// TIA Portal V20 export
// export: Created 2025-12-01T14:57:09.6520783Z, ExportSetting None, DisplayName Totally Integrated Automation Portal, DisplayVersion V20 Update 3, DisplayName TIA Portal Openness, DisplayVersion V20 Update 3, DisplayName TIA Portal Version Control Interface, DisplayVersion V20 Update 3, DisplayName STEP 7 Professional, DisplayVersion V20 Update 3, DisplayName STEP 7 Safety, DisplayVersion V20 Update 2, DisplayName WinCC Basic/Comfort/Advanced, DisplayVersion V20 Update 3, DisplayName WinCC Professional, DisplayVersion V20 Update 3, DisplayName WinCC Unified, DisplayVersion V20 Update 3
FUNCTION "FC722_EliminarUT_DeMesa" : Void   // FC722, LAD
TITLE = EliminarUT_DeMesa - Eliminar la UT de la BD
{ S7_Optimized_Access := 'FALSE' }
AUTHOR : TRACKING
NAME : 20130301
VERSION : 3.0
// stored: AutoNumber false, SetENOAutomatically false
   VAR_INPUT
      NumeroUT : UInt;
   END_VAR
   VAR_TEMP
      Mesa : UInt;   // Mesa
      AnteriorUT : UInt;   // UT Anterior
      SiguienteUT : UInt;   // UT Siguiente
      MckeyTemporal : UDInt;   // Para la ordenacion con Mckey
      ColaMckey : UInt;
      ValorReturn : Int;
      Cero : Byte;
   END_VAR
BEGIN

NETWORK
TITLE = Inicilizar
////////////////////////////////////////////////////////////////////////////////
////////////////////////////////////////////////////////////////////////////////
// Inicializa las variables
      L     0;
      T     #AnteriorUT;
      T     #SiguienteUT;



NETWORK
TITLE = Modificar BD de la Mesa -- Previo
////////////////////////////////////////////////////////////////////////////////
////////////////////////////////////////////////////////////////////////////////
////////////////////////////////////////////////////////////////////////////////
// Datos de la UT Mesa, Anterior UT y Siguiente UT
      L     "DB812_UTs_Control".UT[#NumeroUT].MesaActual;
      L     "CTE_OffsetMesa";
      -I;
      T     #Mesa;

      L     "DB812_UTs_Control".UT[#NumeroUT].UT_AnteriorMesa;
      T     #AnteriorUT;
      L     "DB812_UTs_Control".UT[#NumeroUT].UT_SiguienteMesa;
      T     #SiguienteUT;

      L     "DB812_UTs_Control".UT[#NumeroUT].Mckey;
      T     #MckeyTemporal;



////////////////////////////////////////////////////////////////////////////////
// Limpieza de la UT

      L     0;  // Valor a rellenar
      T     #Cero;

// Borrado del DB de los Datos de la UT
      CALL  FILL
      ( BVAL    := #Cero,
        RET_VAL := #ValorReturn,
        BLK     := "DB812_UTs_Control".UT[#NumeroUT]
      );

// Borrado del DB de la Rutas de la UT
      CALL  FILL
      ( BVAL    := #Cero,
        RET_VAL := #ValorReturn,
        BLK     := "DB813_UTs_Ruta".UT[#NumeroUT]
      );

// Borrado del DB de los Datos Auxiliares de la UT
      CALL  FILL
      ( BVAL    := #Cero,
        RET_VAL := #ValorReturn,
        BLK     := "DB814_UTs_Etiqueta".UT[#NumeroUT]
      );
      CALL  FILL
      ( BVAL    := #Cero,
        RET_VAL := #ValorReturn,
        BLK     := "DB815_UTs_Datos".UT[#NumeroUT]
      );
      CALL  FILL
      ( BVAL    := #Cero,
        RET_VAL := #ValorReturn,
        BLK     := "DB816_UTs_TextoPantalla".UT[#NumeroUT]
      );
      CALL  FILL
      ( BVAL    := #Cero,
        RET_VAL := #ValorReturn,
        BLK     := "DB820_UTs_DatosQUBIQA".UT[#NumeroUT]
      );
      CALL  FILL
      ( BVAL    := #Cero,
        RET_VAL := #ValorReturn,
        BLK     := "DB821_UTs_DatosIKPAL".UT[#NumeroUT]
      );



NETWORK
TITLE = -- UT Anterior
////////////////////////////////////////////////////////////////////////////////
////////////////////////////////////////////////////////////////////////////////
////////////////////////////////////////////////////////////////////////////////
// Modificar la UT Anterior
      SET;
      L     #AnteriorUT;
      L     0;
      ==I;  // Era la UT primera de la Mesa
      JC    PrimeraUT_EnColaMesa;
      JU    NoPrimeraUT_EnColaMesa;


////////////////////////////////////////////////////////////////////////////////
// No es la primar UT de la Mesa
NoPrimeraUT_EnColaMesa:NOP   0;
      L     #SiguienteUT;
      T     "DB812_UTs_Control".UT[#AnteriorUT].UT_SiguienteMesa;

      JU    SiguienteUT_EnColaMesa;


////////////////////////////////////////////////////////////////////////////////
// Es la primera UT de la Mesa
PrimeraUT_EnColaMesa:NOP   0;
      L     #SiguienteUT;
      T     "DB810_ColasMesas".Colas[#Mesa].UT_PrimeraMesa;

      JU    SiguienteUT_EnColaMesa;



NETWORK
TITLE = -- UT Siguiente
////////////////////////////////////////////////////////////////////////////////
////////////////////////////////////////////////////////////////////////////////
////////////////////////////////////////////////////////////////////////////////
// Modificar la UT Siguiente
SiguienteUT_EnColaMesa:NOP   0;
      L     #SiguienteUT;
      L     0;
      ==I;
      JC    Final_EnColaDeMesa;  // Era la UT ultima de la Mesa

////////////////////////////////////////////////////////////////////////////////
// No es la Ultima UT de la Mesa
      L     #AnteriorUT;
      T     "DB812_UTs_Control".UT[#SiguienteUT].UT_AnteriorMesa;

      JU    Final_EnColaDeMesa;



NETWORK
TITLE = -- Final
////////////////////////////////////////////////////////////////////////////////
////////////////////////////////////////////////////////////////////////////////
////////////////////////////////////////////////////////////////////////////////
Final_EnColaDeMesa:NOP   0;



NETWORK
TITLE = Modificar BD de la Ordenacion del Mckey -- Previo
////////////////////////////////////////////////////////////////////////////////
////////////////////////////////////////////////////////////////////////////////
////////////////////////////////////////////////////////////////////////////////
// ----- Antes de acabar eliminar de la ordenacion por Mckey

      L     0;  // Si Mckey es 0
      L     #MckeyTemporal;  // Nunca se ha ordenado por Mckey
      ==D;
      JC    Final_EnColaMckey;  // Ir al final de la ordenacion por Mckey


////////////////////////////////////////////////////////////////////////////////
////////////////////////////////////////////////////////////////////////////////
////////////////////////////////////////////////////////////////////////////////
      L     #MckeyTemporal;
      L     10000;  // Hay 10.000 Colas para el Mckey
      MOD;
      T     #ColaMckey;  // Numero de la Cola del Mckey


      L     "DB811_ColasMckeys".MckeyUT[#NumeroUT].UT_AnteriorMckey;
      T     #AnteriorUT;
      L     "DB811_ColasMckeys".MckeyUT[#NumeroUT].UT_SiguienteMcKey;
      T     #SiguienteUT;

// Limpieza
      L     0;
      T     "DB811_ColasMckeys".MckeyUT[#NumeroUT].UT_AnteriorMckey;
      T     "DB811_ColasMckeys".MckeyUT[#NumeroUT].UT_SiguienteMcKey;



NETWORK
TITLE = -- UT Anterior
////////////////////////////////////////////////////////////////////////////////
////////////////////////////////////////////////////////////////////////////////
////////////////////////////////////////////////////////////////////////////////
// ----- UT Anterior Mckey
      L     #AnteriorUT;
      L     0;
      ==I;  // Esta la primera ??????
      JC    PrimeraUT_EnColaMckey;
      JU    NoPrimeraUT_EnColaMckey;


////////////////////////////////////////////////////////////////////////////////
// ----- No es la primera
NoPrimeraUT_EnColaMckey:NOP   0;
      L     #SiguienteUT;
      T     "DB811_ColasMckeys".MckeyUT[#AnteriorUT].UT_SiguienteMcKey;

      JU    SiguienteUT_EnColaMckey;  // Ir a ordenar la UT siguiente


////////////////////////////////////////////////////////////////////////////////
// ------ Es la Pimera
PrimeraUT_EnColaMckey:NOP   0;
      L     #SiguienteUT;
      T     "DB811_ColasMckeys".Colas_Mckey[#ColaMckey].UT_PrimerMckey;

      JU    SiguienteUT_EnColaMckey;  // Ir a Ordenar la UT siguinete



NETWORK
TITLE = -- UT Siguiente
////////////////////////////////////////////////////////////////////////////////
////////////////////////////////////////////////////////////////////////////////
////////////////////////////////////////////////////////////////////////////////
// ---- UT Siguinete Mckey
SiguienteUT_EnColaMckey:NOP   0;
      L     #SiguienteUT;
      L     0;
      ==I;
      JC    Final_EnColaMckey;  // Esta la ultima ????


////////////////////////////////////////////////////////////////////////////////
/// ---- No ses la Ultima
      L     #AnteriorUT;
      T     "DB811_ColasMckeys".MckeyUT[#SiguienteUT].UT_AnteriorMckey;

      JU    Final_EnColaMckey;  // Ir al final de la ordenacion por Mckey



NETWORK
TITLE = -- Final
////////////////////////////////////////////////////////////////////////////////
////////////////////////////////////////////////////////////////////////////////
////////////////////////////////////////////////////////////////////////////////
// Se acabo la ordenacion

Final_EnColaMckey:NOP   0;




END_FUNCTION
